{attribute 'no_explicit_call' := 'This FB is a CLASS and must be accessed using methods or properties'}
{attribute 'enable_dynamic_creation'}
{attribute 'hide_all_locals'}
FUNCTION_BLOCK FB_DynamicArrayBinary
VAR
	buffer : FB_JsonDynDomParser;
	root : sJsonValue;
END_VAR

PROPERTY PRIVATE _Array : sJsonValue
GET
IF root <> 0 THEN
	_Array := root;
ELSE
	root := buffer.NewDocument();
	_Array := buffer.SetArray(root,0);
END_IF
END_GET
END_PROPERTY

METHOD PUBLIC AddLast : BOOL
VAR_INPUT
	Value : ANY;
END_VAR
AddLast := buffer.PushbackHexBinaryValue(v:= _Array, p := Value.pValue,n := Value.diSize) <> 0;
END_METHOD

METHOD PUBLIC AddStringLast : BOOL
VAR_INPUT
	Value : ANY_STRING;
END_VAR
AddStringLast := buffer.PushbackHexBinaryValue(v:= _Array, p := Value.pValue,n := TO_DINT(LEN2(Value.pValue)+ 1)) <> 0;
END_METHOD

METHOD PUBLIC Clear : BOOL
VAR
	_arrayElement : SJsonAIterator;
END_VAR
_arrayElement := buffer.ArrayBegin(_array);
IF _arrayElement <> 0 THEN
	Clear := buffer.ClearArray(v := _array,i := _arrayElement);
END_IF
END_METHOD

METHOD PUBLIC CopyArrayString : BOOL
VAR_IN_OUT CONSTANT
  	pDoc : STRING; 
END_VAR
VAR_INPUT
	nDoc : UDINT;
END_VAR
CopyArrayString := buffer.copyjson(v:= _Array, pDoc:= pDoc,nDoc := nDoc) <> 0;
END_METHOD

PROPERTY PUBLIC Count : UDINT
GET
Count := buffer.GetArraySize(_array);
END_GET
END_PROPERTY

PROPERTY PUBLIC FirstIndex : UDINT
GET
FirstIndex := 0;
END_GET
END_PROPERTY

PROPERTY PUBLIC LastIndex : UDINT
GET
IF Count = 0 THEN
	LastIndex := 0;
ELSE 
	LastIndex := Count - 1;
END_IF
END_GET
END_PROPERTY

METHOD PUBLIC RemoveFirst : BOOL
VAR
	_arrayElement : SJsonAIterator;
END_VAR
RemoveFirst := TryDeleteIndex(0);
END_METHOD

METHOD PUBLIC RemoveLast: BOOL
VAR
	_arrayElement : SJsonAIterator;
END_VAR
RemoveLast := TryDeleteIndex(LastIndex);
END_METHOD

METHOD PUBLIC TryDeleteIndex : BOOL
VAR_INPUT
	Index : UDINT;
END_VAR
VAR
	_arrayElement : SJsonAIterator;
END_VAR
_arrayElement := buffer.GetArrayValueByIdx(_Array, Index);
IF _arrayElement <> 0 THEN
	TryDeleteIndex := buffer.RemoveArray(v := _array,i := _arrayElement);
END_IF
END_METHOD

METHOD PUBLIC TryGetIndex : BOOL;
VAR_INPUT
	Index : UDINT;
	Destination : ANY;
END_VAR
	TryGetIndex := buffer.GetHexBinary(v:=  buffer.GetArrayValueByIdx(_Array, Index),p := Destination.pValue, n:= Destination.diSize) <> 0;
END_METHOD

METHOD PUBLIC TryGetIndexTo : BOOL;
VAR_INPUT
	Index : UDINT;
	Destination : PVOID;
	DestinationSize : UDINT;
END_VAR
VAR
	_arrayElement : SJsonAIterator;
END_VAR
_arrayElement := buffer.GetArrayValueByIdx(_Array, Index);
IF _arrayElement <> 0 THEN
	TryGetIndexTo := buffer.GetHexBinary(v:= _arrayElement,p := Destination, n:= TO_DINT(DestinationSize)) <> 0;
END_IF
END_METHOD

METHOD PUBLIC TrySetIndex : BOOL
VAR_INPUT
	Index : UDINT;
	Value : ANY;
END_VAR
TrySetIndex := buffer.SetHexBinary(v:= buffer.GetArrayValueByIdx(_Array, Index),p := Value.pValue, n:= Value.diSize) <> 0;
END_METHOD

METHOD PUBLIC TrySetIndexTo : BOOL
VAR_INPUT
	Index : UDINT;
	Value : PVOID;
	ValueSize : UDINT;
END_VAR
VAR
	_arrayElement : SJsonAIterator;
END_VAR
_arrayElement := buffer.GetArrayValueByIdx(_Array, Index);
IF _arrayElement <> 0 THEN
	TrySetIndexTo := buffer.SetHexBinary(v:= _arrayElement,p := Value, n:= TO_DINT(ValueSize)) <> 0;
END_IF
END_METHOD

END_FUNCTION_BLOCK

(* stored: Version 1.1.0.1, ProductVersion 3.1.4024.12
   POU FB_DynamicArrayBinary: Id {bd038ba7-a1bc-47e2-9ed6-417afa2273f3}, SpecialFunc None
   Folder Private: Id {609a49c3-0e57-48e1-8f47-660d6b5240b9}
   Property _Array: Id {2d9b35e8-084d-4a2e-8508-99686a3ca39a}
   Get Get: Id {cddee576-1903-4125-8185-8bb15cadbfa7}
   Method AddLast: Id {e7ce70d9-3b07-44f5-91dd-2c74abe4909a}
   Method AddStringLast: Id {d4c3b84b-444d-48f7-aae9-b19405fd164a}
   Method Clear: Id {2eee8e88-e6c2-42cf-ac7b-53a97395f9e3}
   Method CopyArrayString: Id {50b91631-6b52-4f36-a2a0-7b0f76fb1c7a}
   Property Count: Id {f42a646f-d940-4f66-a7bd-a47e4ecea4e2}
   Get Get: Id {149457ae-80b3-4635-a3b8-88e24670a51e}
   Property FirstIndex: Id {55c40de4-846e-428e-b3aa-c73de79c1c96}
   Get Get: Id {18fb2041-4f7b-4240-9ccc-c025450abd0e}
   Property LastIndex: Id {30f8dfcb-e115-4d0d-8f6c-04af3ae62b68}
   Get Get: Id {e61528ec-832e-4578-9bf1-bb056e838a31}
   Method RemoveFirst: Id {0a80c3ff-b7a1-4969-bb74-e74b4347884d}
   Method RemoveLast: Id {d97db563-80d9-45c9-8257-4ba1366d4144}
   Method TryDeleteIndex: Id {12575d30-50d7-482a-88fc-387d34512a5b}
   Method TryGetIndex: Id {b22fb237-c6a8-4be5-84f7-53ac05df9f3c}
   Method TryGetIndexTo: Id {ba1d405c-bcf2-4886-8698-5263a214e9ed}
   Method TrySetIndex: Id {71be93ee-6a3b-4412-96aa-3d02a5c18350}
   Method TrySetIndexTo: Id {1ffc65df-fc66-4971-bf58-e9fa70b3ba82} *)
